FUNCTION_BLOCK FB_CommandChangeReset EXTENDS FB_CommandChange IMPLEMENTS ITF_CommandChange
VAR

END_VAR

(*			
	EVERDE sp. z o.o.
	Rafał Osajda		03.11.2025		TC 4024.66
	Test czy można zmienić stan lub tryb i zwraca czy można i uruchamia zmianę
*)
METHOD PUBLIC Execute : BOOL
VAR_INPUT
END_VAR
IF (TRUE) THEN
	THIS^.itfSaMController.ChangeStateTo (eNewState := E_SaMStates.Resetting);
END_IF
END_METHOD

METHOD FB_init : BOOL
VAR_INPUT
	bInitRetains : BOOL; // if TRUE, the retain variables are initialized (warm start / cold start)
	bInCopyCode : BOOL;  // if TRUE, the instance afterwards gets moved into the copy code (online change)
END_VAR
THIS^.SetText (eLocation := E_BaseLocation.pl, wsDescription := "Command change state - Reset");
THIS^.SetText (eLocation := E_BaseLocation.en, wsDescription := "Command change state - Reset");
THIS^.SetText (eLocation := E_BaseLocation.de, wsDescription := "Command change state - Reset");
THIS^.SetName (stName := THIS^.GetTexts ());
END_METHOD

END_FUNCTION_BLOCK

(* stored: Version 1.1.0.1
   POU FB_CommandChangeReset: Id {a1007ffe-bcd5-0f21-22f7-0abd1e646a58}, SpecialFunc None
   Method Execute: Id {b1aa8aaa-8518-0852-0151-9ad82e74e41a}
   Method FB_init: Id {1bcce602-1e60-0f12-1637-682824ccb327} *)
